{attribute 'qualified_only'}
{attribute 'strict'}
TYPE Homing :
(
	IDLE,
	
	START,
	RETRY,
	
	STOP,
	SET,
	DONE,
	
	size
);
END_TYPE
(*
general homing sequence:
	on drive.homingSequence() call, home towards home sensor
	if home reached, set position and finish homing as usual
	if outer limit reached, traverse towards inner limit
		when inner limit reached, retry homing
*)

(* stored: Version 1.1.0.1, ProductVersion 3.1.4024.11
   DUT Homing: Id {8cb9de35-a383-425e-8ca1-d663d47beaf0} *)
